// TIA Portal V20 export
// export: Created 2025-12-01T14:57:27.001075Z, ExportSetting None, DisplayName Totally Integrated Automation Portal, DisplayVersion V20 Update 3, DisplayName TIA Portal Openness, DisplayVersion V20 Update 3, DisplayName TIA Portal Version Control Interface, DisplayVersion V20 Update 3, DisplayName STEP 7 Professional, DisplayVersion V20 Update 3, DisplayName STEP 7 Safety, DisplayVersion V20 Update 2, DisplayName WinCC Basic/Comfort/Advanced, DisplayVersion V20 Update 3, DisplayName WinCC Professional, DisplayVersion V20 Update 3, DisplayName WinCC Unified, DisplayVersion V20 Update 3
FUNCTION "FC607_Estado_Peines" : Void   // FC607, LAD
{ S7_Optimized_Access := 'TRUE' }
// stored: AutoNumber false, SetENOAutomatically false
   VAR_INPUT
      ID_Quimarox : UInt;
   END_VAR
   VAR_OUTPUT
      VaciosPeines : Bool;
   END_VAR
   VAR_TEMP
      Maximo_peines : UInt;
      Contador_auxiliar : UInt;
   END_VAR
BEGIN

NETWORK
TITLE = Inicializar
      L     "DB600_ConfigQuimarox".Quimarox[#ID_Quimarox].datos_config.Numero_vagones;
      T     #Maximo_peines;



NETWORK
TITLE = Busqueda de Vagones cargados
      L     1;
      T     #Contador_auxiliar;

      SET;
      =     #VaciosPeines;

Bucle:NOP   0;

      SET;
      AN    "DB601_PeinesQuimarox".Quimarox[#ID_Quimarox].vagon[#Contador_auxiliar].Carrier_Cargado;
      JC    siguiente;


      CLR;
      =     #VaciosPeines;
      BE;  // NO hace falta mirar mas, hay carga

siguiente:NOP   0;

      SET;
      L     #Contador_auxiliar;
      L     #Maximo_peines;
      ==I;
      JC    fin;


      L     #Contador_auxiliar;
      L     1;
      +I;
      T     #Contador_auxiliar;

      JU    Bucle;

fin:  BE;  // Fin de la Funcion
END_FUNCTION
